{attribute 'qualified_only'}
{attribute 'strict'}
{attribute 'to_string'}
TYPE eControlSources :
(
	Local 				:= 0,
	ExternalController 	:= 1,
	PowerNet			:= 2	
);
END_TYPE

(* stored: Version 1.1.0.1, ProductVersion 3.1.4026.18
   DUT eControlSources: Id {8ced42d4-d5f6-424e-917d-528f9475ba7d} *)
